// TIA Portal V17 export
// export: Created 2023-05-07T12:12:22.7639653Z, ExportSetting WithDefaults, DisplayName Totally Integrated Automation Portal, DisplayVersion V17, DisplayName TIA Portal Openness, DisplayVersion V17, DisplayName TIA Portal Version Control Interface, DisplayVersion V17, DisplayName TIA Portal Test Suite Advanced, DisplayVersion V17, DisplayName STEP 7 Professional, DisplayVersion V17, DisplayName SIMATIC Energy Suite, DisplayVersion V17, DisplayName STEP 7 Safety, DisplayVersion V17, DisplayName WinCC Professional, DisplayVersion V17
DATA_BLOCK "Generator_DB"   // DB14
VERSION : 0.1
// stored: AutoNumber true, InstanceOfName Generator, InstanceOfType FB
"Generator"
   // VAR_OUTPUT
   //    wartosc_zaklocenia : Real;
   //    u : LReal;
   // END_VAR
   // VAR
   //    k : Real;
   //    i : Int;
   // END_VAR
BEGIN
END_DATA_BLOCK
